SYSTEM Test Reader
  (* Version 1.0, 2005-06-27, Goran Cengic, Chalmers *)
  DEVICE Test Device : DeviceType_not_used
    RESOURCE TestResource : ResourceType_not_used
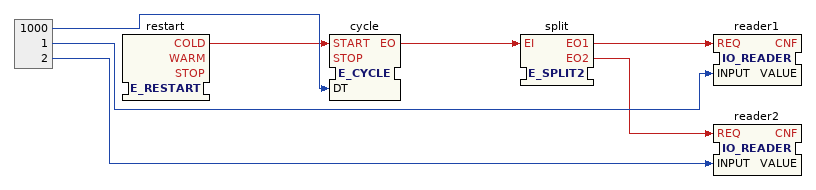
      FBS
        restart : E_RESTART;
        cycle : E_CYCLE;
        split : E_SPLIT2;
        reader1 : IO_READER;
        reader2 : IO_READER;
      END_FBS
      EVENT_CONNECTIONS
        restart.COLD TO cycle.START;
        cycle.EO TO split.EI;
        split.EO1 TO reader1.REQ;
        split.EO2 TO reader2.REQ;
      END_CONNECTIONS
      DATA_CONNECTIONS
        1000 TO cycle.DT;
        1 TO reader1.INPUT;
        2 TO reader2.INPUT;
      END_CONNECTIONS
    END_RESOURCE
  END_DEVICE
END_SYSTEM
